SUBAPPLICATION Motor (* Subapplication Type *)
  (* Standard: 61499-2 *)
  (* Version 1.0, 2018-09-13, az *)
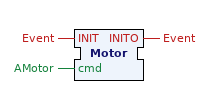
  EVENT_INPUT
    INIT;
  END_EVENT
  EVENT_OUTPUT
    INITO;
  END_EVENT
  SOCKETS
    cmd : AMotor;
  END_SOCKETS
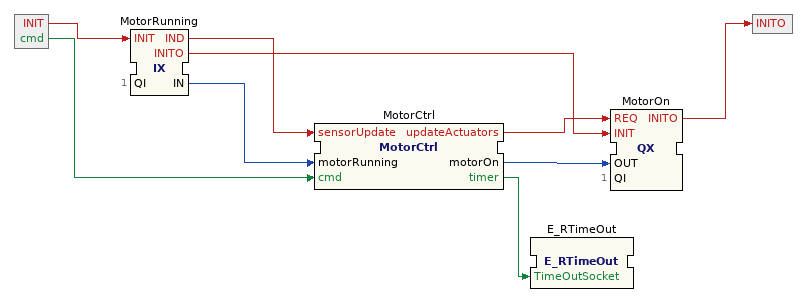
  FBS
    MotorRunning : IX(QI := 1);
    MotorOn : QX(QI := 1);
    MotorCtrl : MotorCtrl;
    E_RTimeOut : E_RTimeOut;
  END_FBS
  EVENT_CONNECTIONS
    MotorRunning.IND TO MotorCtrl.sensorUpdate;
    MotorCtrl.updateActuators TO MotorOn.REQ;
    INIT TO MotorRunning.INIT;
    MotorRunning.INITO TO MotorOn.INIT;
    MotorOn.INITO TO INITO;
  END_CONNECTIONS
  DATA_CONNECTIONS
    MotorRunning.IN TO MotorCtrl.motorRunning;
    MotorCtrl.motorOn TO MotorOn.OUT;
  END_CONNECTIONS
  ADAPTER_CONNECTIONS
    cmd TO MotorCtrl.cmd;
    MotorCtrl.timer TO E_RTimeOut.TimeOutSocket;
  END_CONNECTIONS
END_SUBAPPLICATION
